FUNCTION_BLOCK PAEActDosingSlider EXTENDS PAEActuator1way_3pos
VAR_INPUT
END_VAR
VAR_OUTPUT
END_VAR
VAR
END_VAR

METHOD PUBLIC PAEActDosingSlider
VAR_INPUT
END_VAR
END_METHOD

END_FUNCTION_BLOCK

(* stored: Version 1.1.0.1, ProductVersion 3.1.4020.12
   POU PAEActDosingSlider: Id {8f801670-1eea-483e-b4cb-65459fc4ad68}, SpecialFunc None
   Method PAEActDosingSlider: Id {f74ffb5a-e9f6-46c8-a11d-c81119b835d4} *)
